// Mitsubishi GX Developer project: PLC_PCO520L2   PLC: Q06UDEH   RS485 Communication Modbus RTU

PROGRAM SP790_RS
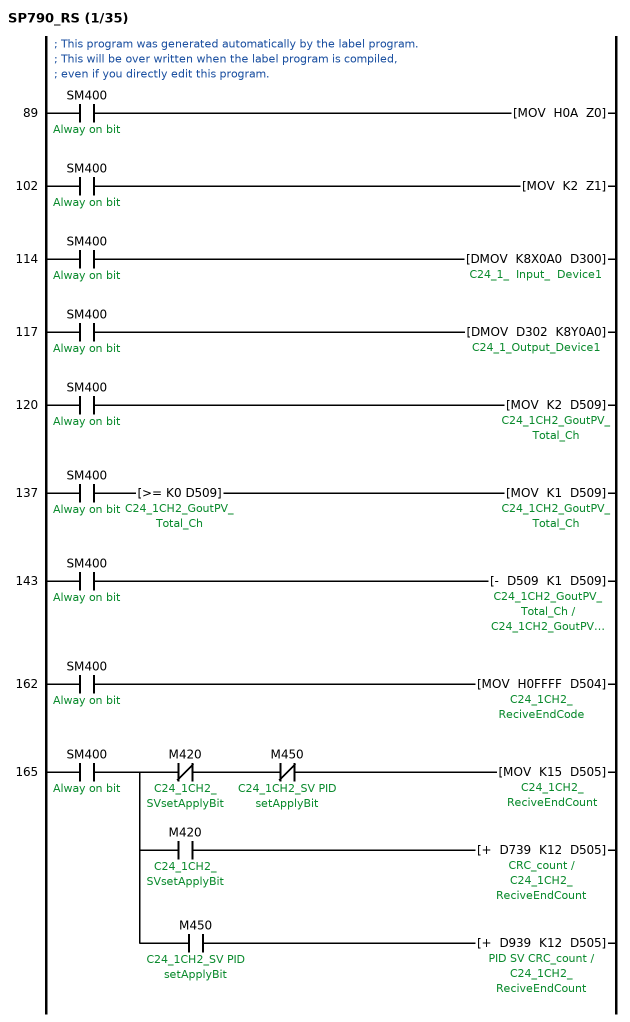
; This program was generated automatically by the label program.
; This will be over written when the label program is compiled,
; even if you directly edit this program.
89    LD      SM400  ; Alway on bit
      MOV     H0A Z0
        [note] Module IO Number
102   LD      SM400  ; Alway on bit
      MOV     K2 Z1
        [note] Channel Number
114   LD      SM400  ; Alway on bit
      DMOV    K8X0A0 D300  ; CH1 Transmission normal completi / C24_1_  Input_  Device1
117   LD      SM400  ; Alway on bit
      DMOV    D302 K8Y0A0  ; C24_1_Output_Device1 / CH1 Transmission request
120   LD      SM400  ; Alway on bit
      MOV     K2 D509  ; C24_1CH2_GoutPV_Total_Ch
        [note] Controller Channel Count
137   LD      SM400  ; Alway on bit
      AND>=   K0 D509  ; C24_1CH2_GoutPV_Total_Ch
      MOV     K1 D509
143   LD      SM400  ; Alway on bit
      -       D509 K1 D509
        [note] Controller Channel Count
162   LD      SM400  ; Alway on bit
      MOV     H0FFFF D504  ; C24_1CH2_ReciveEndCode
165   LD      SM400  ; Alway on bit
      MPS
      ANI     M420  ; C24_1CH2_SVsetApplyBit
      ANI     M450  ; C24_1CH2_SV PID setApplyBit
      MOV     K15 D505  ; C24_1CH2_ReciveEndCount
      MRD
      AND     M420  ; C24_1CH2_SVsetApplyBit
      +       D739 K12 D505  ; CRC_count
      MPP
      AND     M450  ; C24_1CH2_SV PID setApplyBit
      +       D939 K12 D505  ; PID SV CRC_count
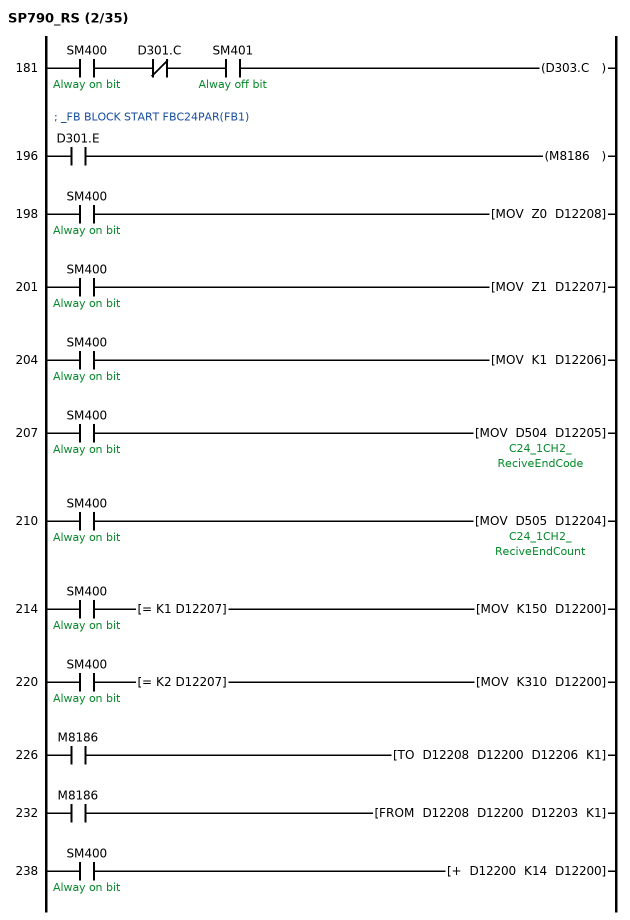
181   LD      SM400  ; Alway on bit
      ANI     D301.C
      AND     SM401  ; Alway off bit
      OUT     D303.C
        [note] System汲沥檬扁拳
; _FB BLOCK START FBC24PAR(FB1)
196   LD      D301.E
      OUT     M8186
198   LD      SM400  ; Alway on bit
      MOV     Z0 D12208
201   LD      SM400  ; Alway on bit
      MOV     Z1 D12207
204   LD      SM400  ; Alway on bit
      MOV     K1 D12206
207   LD      SM400  ; Alway on bit
      MOV     D504 D12205
210   LD      SM400  ; Alway on bit
      MOV     D505 D12204
; FB START
214   LD      SM400  ; Alway on bit
      AND=    K1 D12207
      MOV     K150 D12200
220   LD      SM400  ; Alway on bit
      AND=    K2 D12207
      MOV     K310 D12200
226   LD      M8186
      TO      D12208 D12200 D12206 K1
232   LD      M8186
      FROM    D12208 D12200 D12203 K1
238   LD      SM400  ; Alway on bit
      +       D12200 K14 D12200
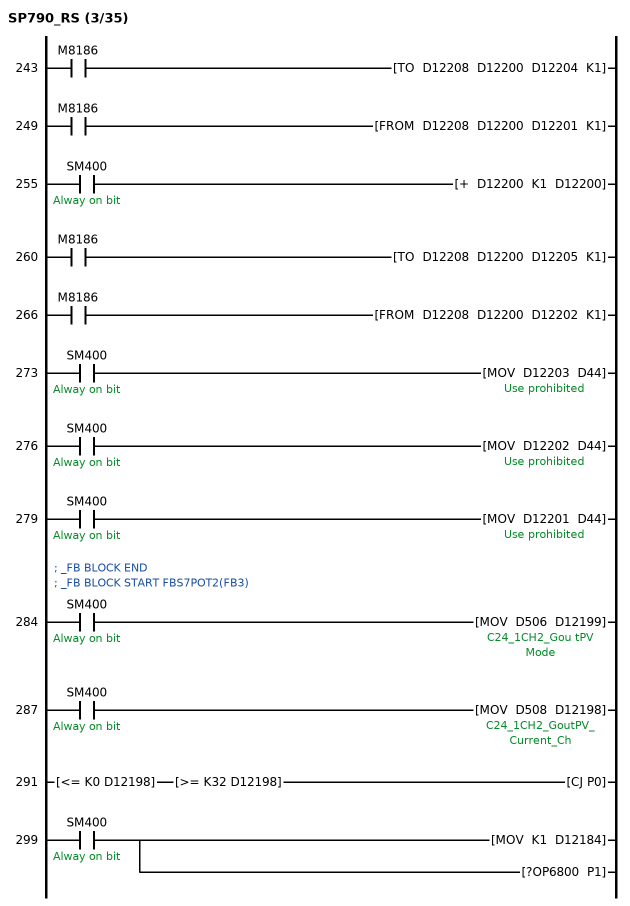
243   LD      M8186
      TO      D12208 D12200 D12204 K1
249   LD      M8186
      FROM    D12208 D12200 D12201 K1
255   LD      SM400  ; Alway on bit
      +       D12200 K1 D12200
260   LD      M8186
      TO      D12208 D12200 D12205 K1
266   LD      M8186
      FROM    D12208 D12200 D12202 K1
; FB END
273   LD      SM400  ; Alway on bit
      MOV     D12203 D44  ; Use prohibited
276   LD      SM400  ; Alway on bit
      MOV     D12202 D44
279   LD      SM400  ; Alway on bit
      MOV     D12201 D44
; _FB BLOCK END
; _FB BLOCK START FBS7POT2(FB3)
284   LD      SM400  ; Alway on bit
      MOV     D506 D12199  ; C24_1CH2_Gou tPV Mode
287   LD      SM400  ; Alway on bit
      MOV     D508 D12198  ; C24_1CH2_GoutPV_Current_Ch
; FB START
291   LD<=    K0 D12198
      AND>=   K32 D12198
      CJ      P0
299   LD      SM400  ; Alway on bit
      MOV     K1 D12184
      ?OP6800 P1
      P0
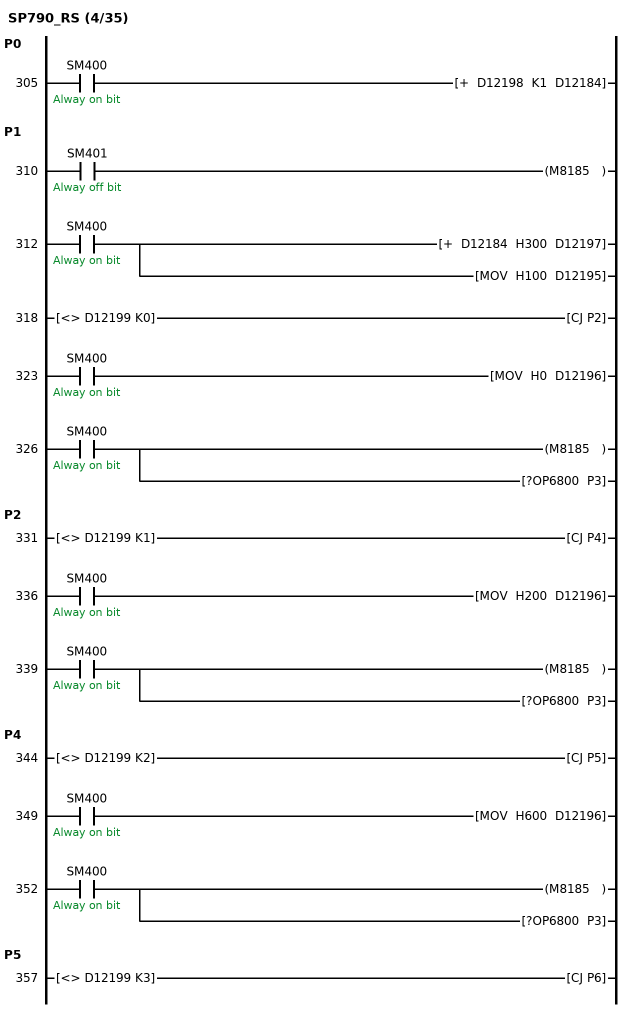
305   LD      SM400  ; Alway on bit
      +       D12198 K1 D12184
      P1
310   LD      SM401  ; Alway off bit
      OUT     M8185
312   LD      SM400  ; Alway on bit
      +       D12184 H300 D12197
      MOV     H100 D12195
318   LD<>    D12199 K0
      CJ      P2
323   LD      SM400  ; Alway on bit
      MOV     H0 D12196
326   LD      SM400  ; Alway on bit
      OUT     M8185
      ?OP6800 P3
      P2
331   LD<>    D12199 K1
      CJ      P4
336   LD      SM400  ; Alway on bit
      MOV     H200 D12196
339   LD      SM400  ; Alway on bit
      OUT     M8185
      ?OP6800 P3
      P4
344   LD<>    D12199 K2
      CJ      P5
349   LD      SM400  ; Alway on bit
      MOV     H600 D12196
352   LD      SM400  ; Alway on bit
      OUT     M8185
      ?OP6800 P3
      P5
357   LD<>    D12199 K3
      CJ      P6
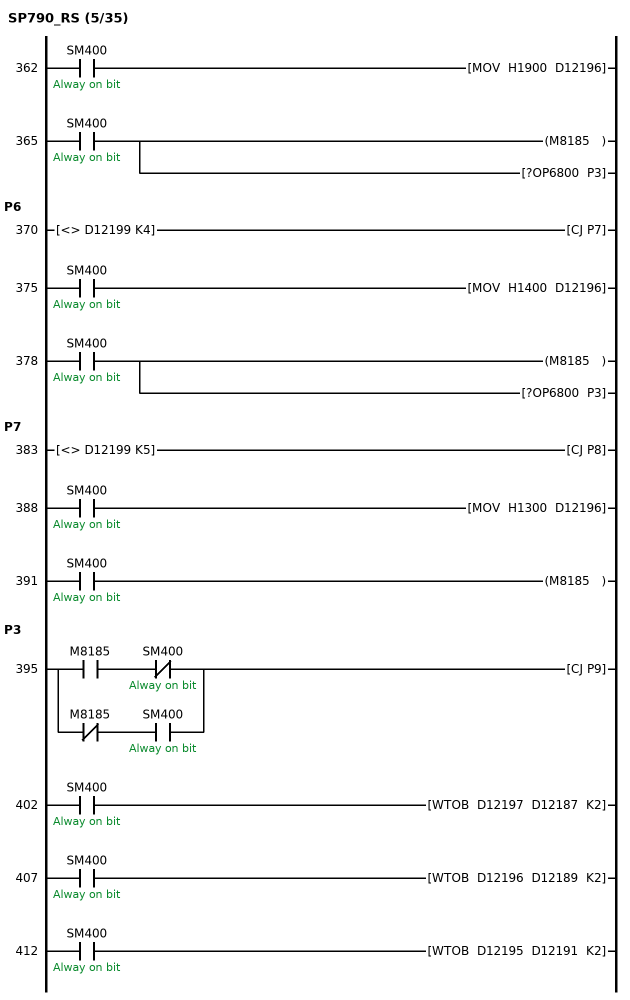
362   LD      SM400  ; Alway on bit
      MOV     H1900 D12196
365   LD      SM400  ; Alway on bit
      OUT     M8185
      ?OP6800 P3
      P6
370   LD<>    D12199 K4
      CJ      P7
375   LD      SM400  ; Alway on bit
      MOV     H1400 D12196
378   LD      SM400  ; Alway on bit
      OUT     M8185
      ?OP6800 P3
      P7
383   LD<>    D12199 K5
      CJ      P8
388   LD      SM400  ; Alway on bit
      MOV     H1300 D12196
391   LD      SM400  ; Alway on bit
      OUT     M8185
      P8
      P3
395   LD      M8185
      ANI     SM400  ; Alway on bit
      LDI     M8185
      AND     SM400  ; Alway on bit
      ORB
      CJ      P9
402   LD      SM400  ; Alway on bit
      WTOB    D12197 D12187 K2
407   LD      SM400  ; Alway on bit
      WTOB    D12196 D12189 K2
412   LD      SM400  ; Alway on bit
      WTOB    D12195 D12191 K2
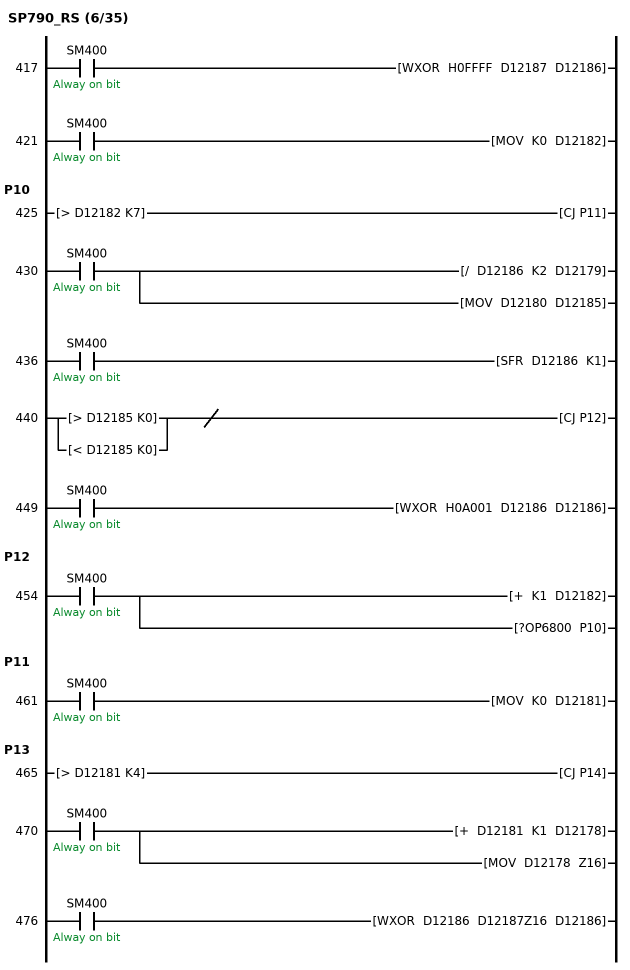
417   LD      SM400  ; Alway on bit
      WXOR    H0FFFF D12187 D12186
421   LD      SM400  ; Alway on bit
      MOV     K0 D12182
      P10
425   LD>     D12182 K7
      CJ      P11
430   LD      SM400  ; Alway on bit
      /       D12186 K2 D12179
      MOV     D12180 D12185
436   LD      SM400  ; Alway on bit
      SFR     D12186 K1
440   LD>     D12185 K0
      OR<     D12185 K0
      INV
      CJ      P12
449   LD      SM400  ; Alway on bit
      WXOR    H0A001 D12186 D12186
      P12
454   LD      SM400  ; Alway on bit
      +       K1 D12182
      ?OP6800 P10
      P11
461   LD      SM400  ; Alway on bit
      MOV     K0 D12181
      P13
465   LD>     D12181 K4
      CJ      P14
470   LD      SM400  ; Alway on bit
      +       D12181 K1 D12178
      MOV     D12178 Z16
476   LD      SM400  ; Alway on bit
      WXOR    D12186 D12187Z16 D12186
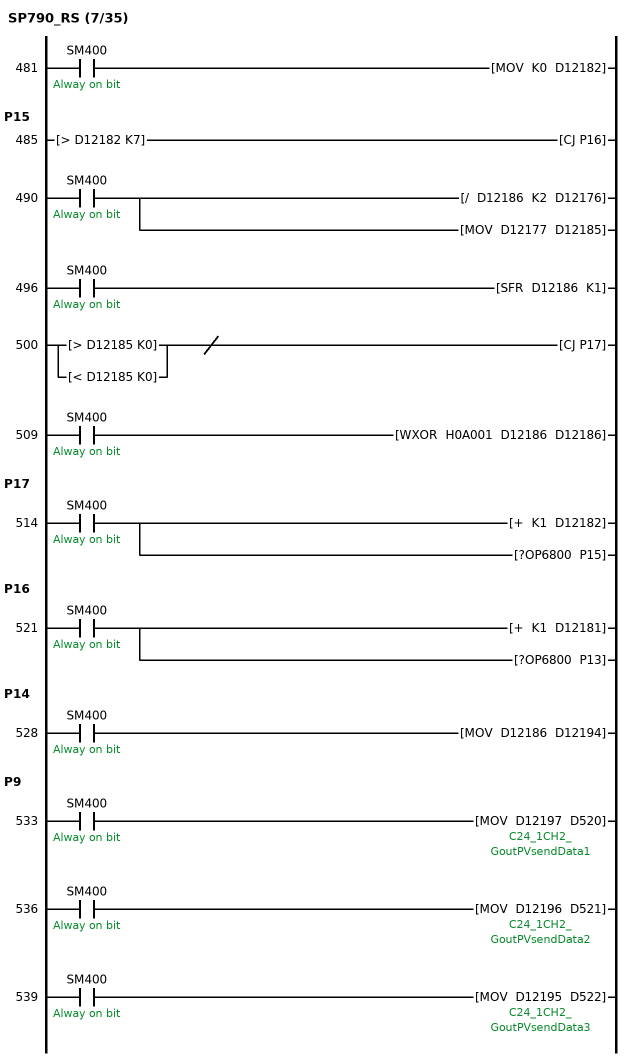
481   LD      SM400  ; Alway on bit
      MOV     K0 D12182
      P15
485   LD>     D12182 K7
      CJ      P16
490   LD      SM400  ; Alway on bit
      /       D12186 K2 D12176
      MOV     D12177 D12185
496   LD      SM400  ; Alway on bit
      SFR     D12186 K1
500   LD>     D12185 K0
      OR<     D12185 K0
      INV
      CJ      P17
509   LD      SM400  ; Alway on bit
      WXOR    H0A001 D12186 D12186
      P17
514   LD      SM400  ; Alway on bit
      +       K1 D12182
      ?OP6800 P15
      P16
521   LD      SM400  ; Alway on bit
      +       K1 D12181
      ?OP6800 P13
      P14
528   LD      SM400  ; Alway on bit
      MOV     D12186 D12194
      P9
; FB END
533   LD      SM400  ; Alway on bit
      MOV     D12197 D520  ; C24_1CH2_GoutPVsendData1
536   LD      SM400  ; Alway on bit
      MOV     D12196 D521  ; C24_1CH2_GoutPVsendData2
539   LD      SM400  ; Alway on bit
      MOV     D12195 D522  ; C24_1CH2_GoutPVsendData3
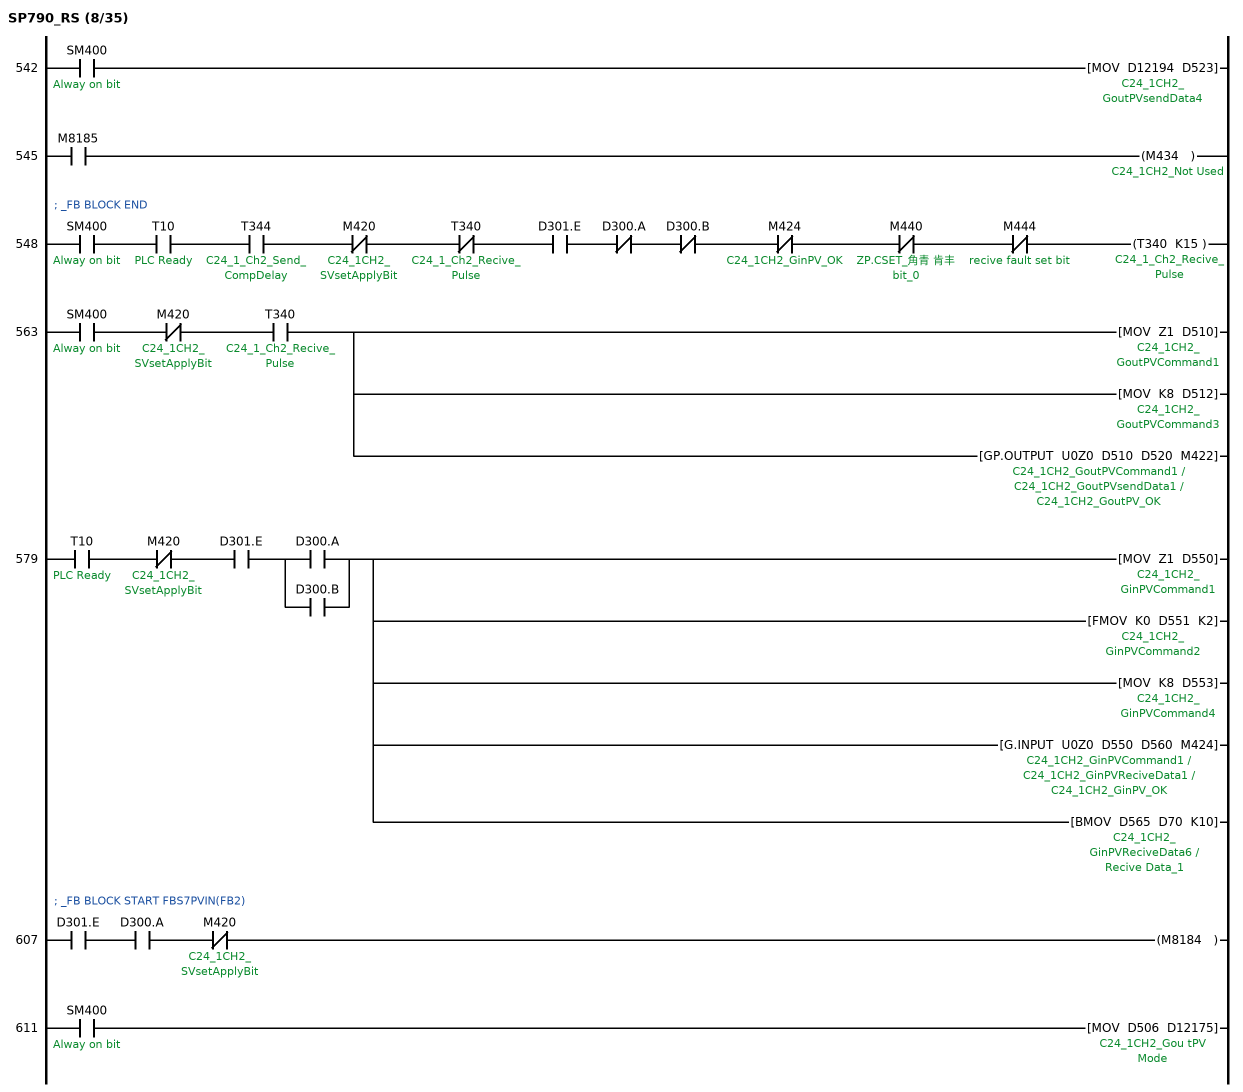
542   LD      SM400  ; Alway on bit
      MOV     D12194 D523  ; C24_1CH2_GoutPVsendData4
545   LD      M8185
      OUT     M434  ; C24_1CH2_Not Used
; _FB BLOCK END
548   LD      SM400  ; Alway on bit
      AND     T10  ; PLC Ready
      AND     T344  ; C24_1_Ch2_Send_CompDelay
      ANI     M420  ; C24_1CH2_SVsetApplyBit
      ANI     T340  ; C24_1_Ch2_Recive_Pulse
      AND     D301.E
      ANI     D300.A
      ANI     D300.B
      ANI     M424  ; C24_1CH2_GinPV_OK
      ANI     M440  ; ZP.CSET_角青 肯丰 bit_0
      ANI     M444  ; recive fault set bit
      OUTH    T340 K15  ; C24_1_Ch2_Recive_Pulse
563   LD      SM400  ; Alway on bit
      ANI     M420  ; C24_1CH2_SVsetApplyBit
      AND     T340  ; C24_1_Ch2_Recive_Pulse
      MOV     Z1 D510  ; C24_1CH2_GoutPVCommand1
      MOV     K8 D512  ; C24_1CH2_GoutPVCommand3
      GP.OUTPUT U0Z0 D510 D520 M422  ; C24_1CH2_GoutPV_OK
579   LD      T10  ; PLC Ready
      ANI     M420  ; C24_1CH2_SVsetApplyBit
      AND     D301.E
      LD      D300.A
      OR      D300.B
      ANB
      MOV     Z1 D550  ; C24_1CH2_GinPVCommand1
      FMOV    K0 D551 K2  ; C24_1CH2_GinPVCommand2
      MOV     K8 D553  ; C24_1CH2_GinPVCommand4
      G.INPUT U0Z0 D550 D560 M424  ; C24_1CH2_GinPVReciveData1
      BMOV    D565 D70 K10  ; C24_1CH2_GinPVReciveData6 / Recive Data_1
; _FB BLOCK START FBS7PVIN(FB2)
607   LD      D301.E
      AND     D300.A
      ANI     M420  ; C24_1CH2_SVsetApplyBit
      OUT     M8184
611   LD      SM400  ; Alway on bit
      MOV     D506 D12175
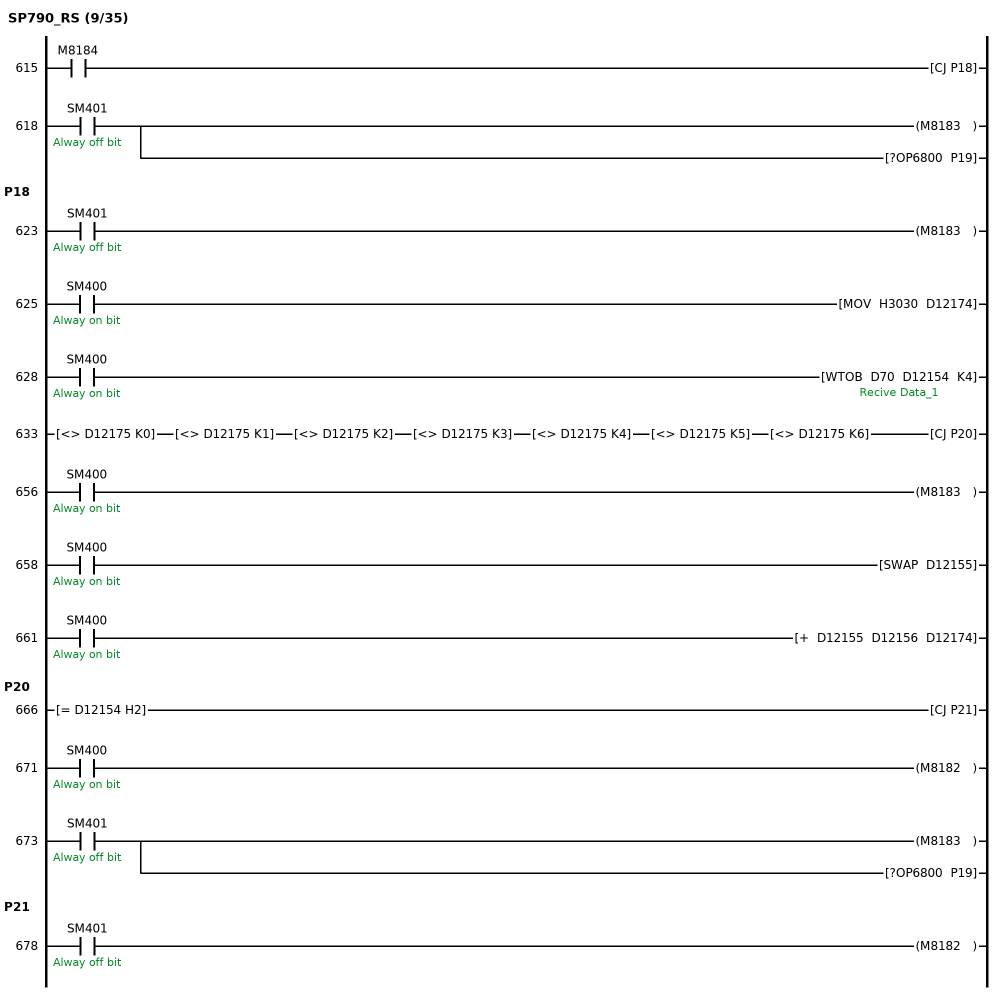
; FB START
615   LD      M8184
      CJ      P18
618   LD      SM401  ; Alway off bit
      OUT     M8183
      ?OP6800 P19
      P18
623   LD      SM401  ; Alway off bit
      OUT     M8183
625   LD      SM400  ; Alway on bit
      MOV     H3030 D12174
628   LD      SM400  ; Alway on bit
      WTOB    D70 D12154 K4
633   LD<>    D12175 K0
      AND<>   D12175 K1
      AND<>   D12175 K2
      AND<>   D12175 K3
      AND<>   D12175 K4
      AND<>   D12175 K5
      AND<>   D12175 K6
      CJ      P20
656   LD      SM400  ; Alway on bit
      OUT     M8183
658   LD      SM400  ; Alway on bit
      SWAP    D12155
661   LD      SM400  ; Alway on bit
      +       D12155 D12156 D12174
      P20
666   LD=     D12154 H2
      CJ      P21
671   LD      SM400  ; Alway on bit
      OUT     M8182
673   LD      SM401  ; Alway off bit
      OUT     M8183
      ?OP6800 P19
      P21
678   LD      SM401  ; Alway off bit
      OUT     M8182
      P19
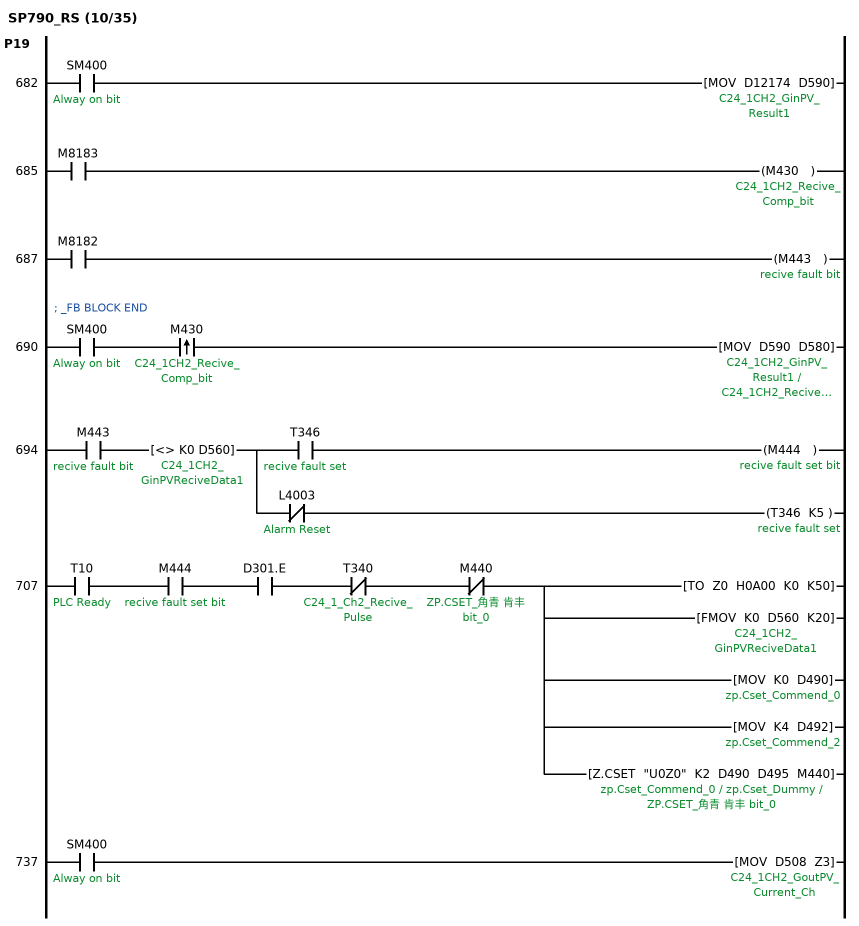
; FB END
682   LD      SM400  ; Alway on bit
      MOV     D12174 D590  ; C24_1CH2_GinPV_Result1
685   LD      M8183
      OUT     M430  ; C24_1CH2_Recive_Comp_bit
687   LD      M8182
      OUT     M443  ; recive fault bit
; _FB BLOCK END
690   LD      SM400  ; Alway on bit
      ANDP    M430  ; C24_1CH2_Recive_Comp_bit
      MOV     D590 D580  ; C24_1CH2_Recive_Value_1
694   LD      M443  ; recive fault bit
      AND<>   K0 D560  ; C24_1CH2_GinPVReciveData1
      MPS
      AND     T346  ; recive fault set
      OUT     M444  ; recive fault set bit
      MPP
      ANI     L4003  ; Alarm Reset
      OUT     T346 K5  ; recive fault set
707   LD      T10  ; PLC Ready
      AND     M444  ; recive fault set bit
      AND     D301.E
      ANI     T340  ; C24_1_Ch2_Recive_Pulse
      ANI     M440  ; ZP.CSET_角青 肯丰 bit_0
      TO      Z0 H0A00 K0 K50
      FMOV    K0 D560 K20
      MOV     K0 D490  ; zp.Cset_Commend_0
      MOV     K4 D492  ; zp.Cset_Commend_2
      Z.CSET  "U0Z0" K2 D490 D495 M440  ; zp.Cset_Dummy
737   LD      SM400  ; Alway on bit
      MOV     D508 Z3
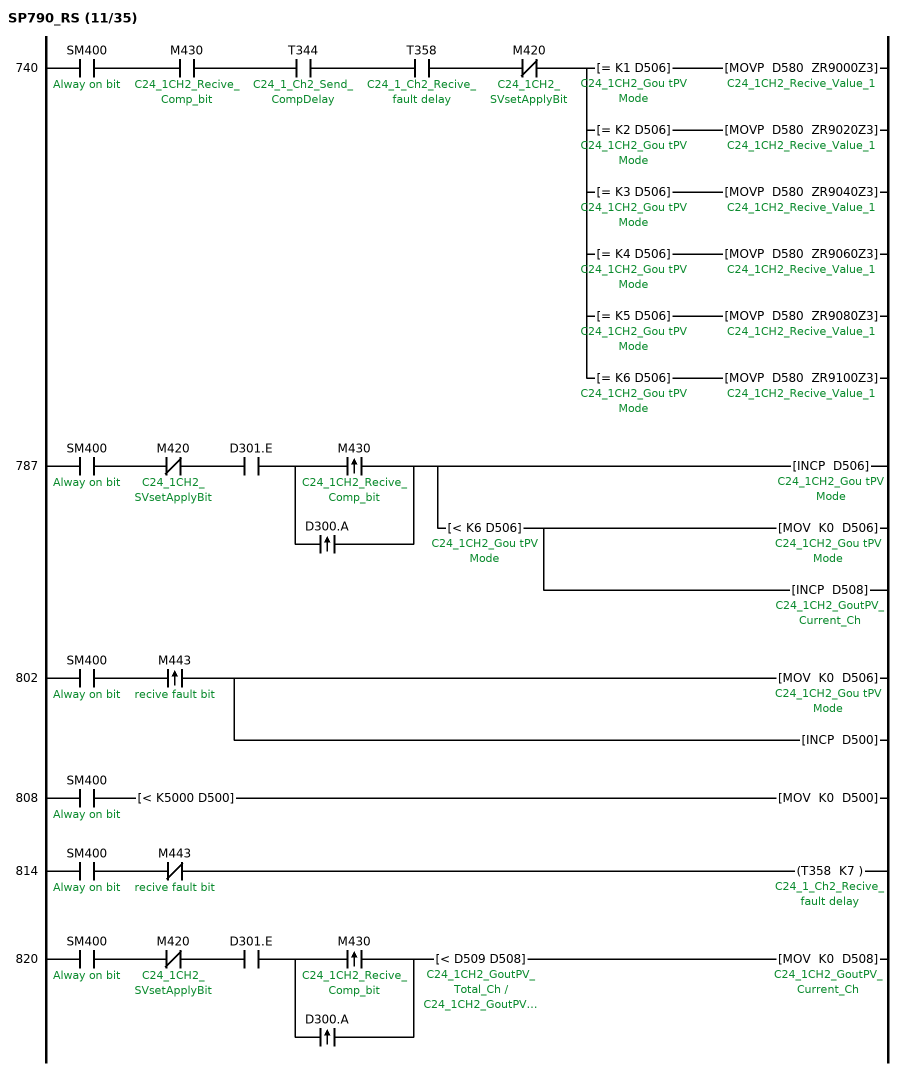
740   LD      SM400  ; Alway on bit
      AND     M430  ; C24_1CH2_Recive_Comp_bit
      AND     T344  ; C24_1_Ch2_Send_CompDelay
      AND     T358  ; C24_1_Ch2_Recive_fault delay
      ANI     M420  ; C24_1CH2_SVsetApplyBit
      MPS
      AND=    K1 D506  ; C24_1CH2_Gou tPV Mode
      MOVP    D580 ZR9000Z3
      MRD
      AND=    K2 D506  ; C24_1CH2_Gou tPV Mode
      MOVP    D580 ZR9020Z3
      MRD
      AND=    K3 D506  ; C24_1CH2_Gou tPV Mode
      MOVP    D580 ZR9040Z3
      MRD
      AND=    K4 D506  ; C24_1CH2_Gou tPV Mode
      MOVP    D580 ZR9060Z3
      MRD
      AND=    K5 D506  ; C24_1CH2_Gou tPV Mode
      MOVP    D580 ZR9080Z3
      MPP
      AND=    K6 D506  ; C24_1CH2_Gou tPV Mode
      MOVP    D580 ZR9100Z3
787   LD      SM400  ; Alway on bit
      ANI     M420  ; C24_1CH2_SVsetApplyBit
      AND     D301.E
      LDP     M430  ; C24_1CH2_Recive_Comp_bit
      ORP     D300.A
      ANB
      INCP    D506
      AND<    K6 D506  ; C24_1CH2_Gou tPV Mode
      MOV     K0 D506
      INCP    D508
802   LD      SM400  ; Alway on bit
      ANDP    M443  ; recive fault bit
      MOV     K0 D506
      INCP    D500
808   LD      SM400  ; Alway on bit
      AND<    K5000 D500
      MOV     K0 D500
814   LD      SM400  ; Alway on bit
      ANI     M443  ; recive fault bit
      OUT     T358 K7  ; C24_1_Ch2_Recive_fault delay
820   LD      SM400  ; Alway on bit
      ANI     M420  ; C24_1CH2_SVsetApplyBit
      AND     D301.E
      LDP     M430  ; C24_1CH2_Recive_Comp_bit
      ORP     D300.A
      ANB
      AND<    D509 D508  ; C24_1CH2_GoutPV_Total_Ch / C24_1CH2_GoutPV_Current_Ch
      MOV     K0 D508
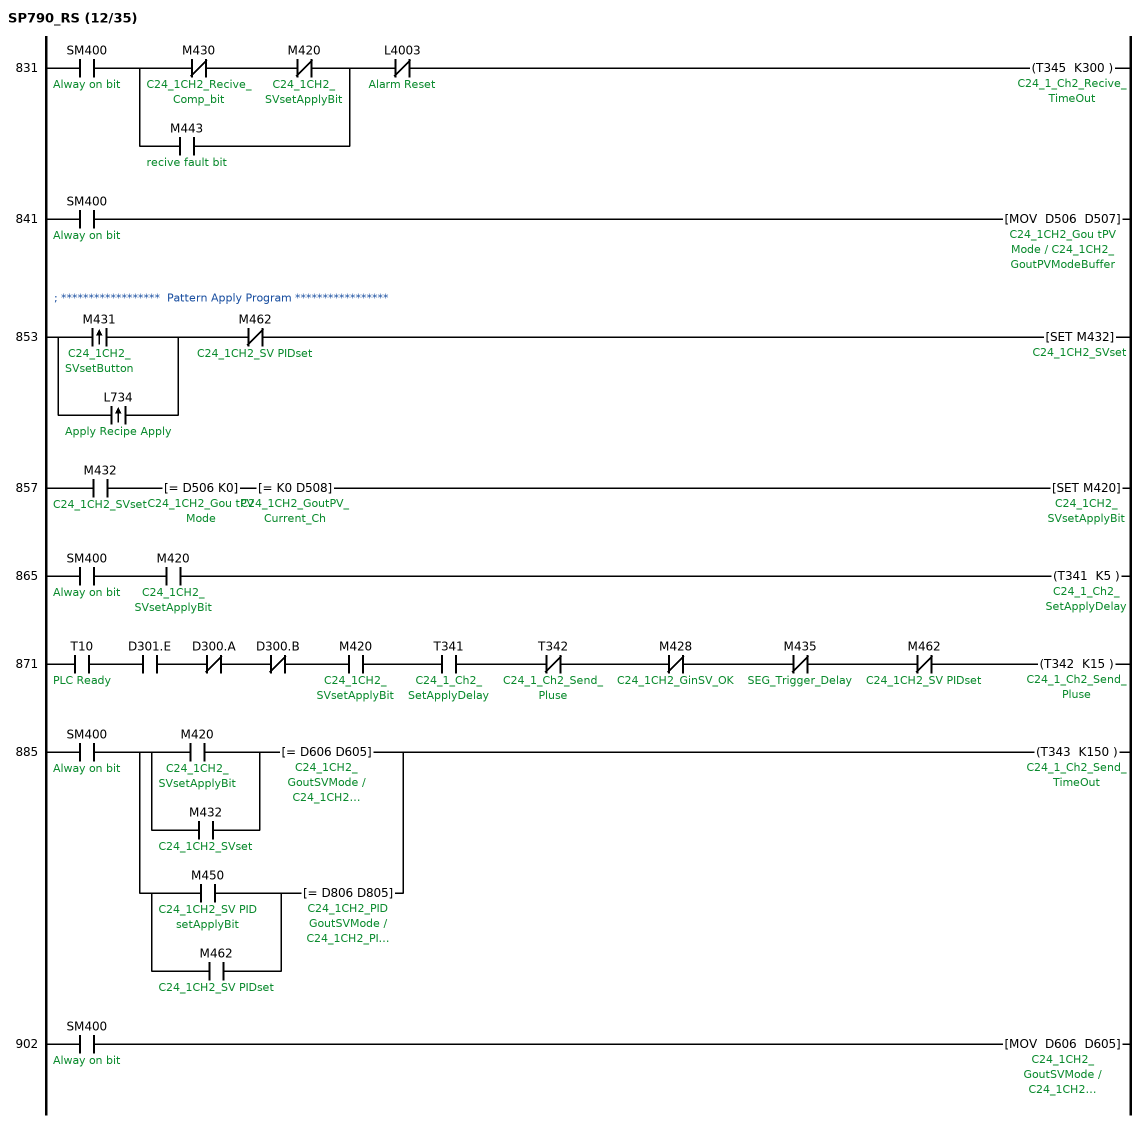
831   LD      SM400  ; Alway on bit
      LDI     M430  ; C24_1CH2_Recive_Comp_bit
      ANI     M420  ; C24_1CH2_SVsetApplyBit
      OR      M443  ; recive fault bit
      ANB
      ANI     L4003  ; Alarm Reset
      OUT     T345 K300  ; C24_1_Ch2_Recive_TimeOut
841   LD      SM400  ; Alway on bit
      MOV     D506 D507  ; C24_1CH2_GoutPVModeBuffer
; 
; 
; 
; 
; ******************  Pattern Apply Program *****************
853   LDP     M431  ; C24_1CH2_SVsetButton
      ORP     L734  ; Apply Recipe Apply
      ANI     M462  ; C24_1CH2_SV PIDset
      SET     M432  ; C24_1CH2_SVset
857   LD      M432  ; C24_1CH2_SVset
      AND=    D506 K0  ; C24_1CH2_Gou tPV Mode
      AND=    K0 D508  ; C24_1CH2_GoutPV_Current_Ch
      SET     M420  ; C24_1CH2_SVsetApplyBit
865   LD      SM400  ; Alway on bit
      AND     M420  ; C24_1CH2_SVsetApplyBit
      OUT     T341 K5  ; C24_1_Ch2_SetApplyDelay
871   LD      T10  ; PLC Ready
      AND     D301.E
      ANI     D300.A
      ANI     D300.B
      AND     M420  ; C24_1CH2_SVsetApplyBit
      AND     T341  ; C24_1_Ch2_SetApplyDelay
      ANI     T342  ; C24_1_Ch2_Send_Pluse
      ANI     M428  ; C24_1CH2_GinSV_OK
      ANI     M435  ; SEG_Trigger_Delay
      ANI     M462  ; C24_1CH2_SV PIDset
      OUTH    T342 K15  ; C24_1_Ch2_Send_Pluse
885   LD      SM400  ; Alway on bit
      LD      M420  ; C24_1CH2_SVsetApplyBit
      OR      M432  ; C24_1CH2_SVset
      AND=    D606 D605  ; C24_1CH2_GoutSVMode / C24_1CH2_ModeBuffer
      LD      M450  ; C24_1CH2_SV PID setApplyBit
      OR      M462  ; C24_1CH2_SV PIDset
      AND=    D806 D805  ; C24_1CH2_PID GoutSVMode / C24_1CH2_PID ModeBuffer
      ORB
      ANB
      OUT     T343 K150  ; C24_1_Ch2_Send_TimeOut
902   LD      SM400  ; Alway on bit
      MOV     D606 D605
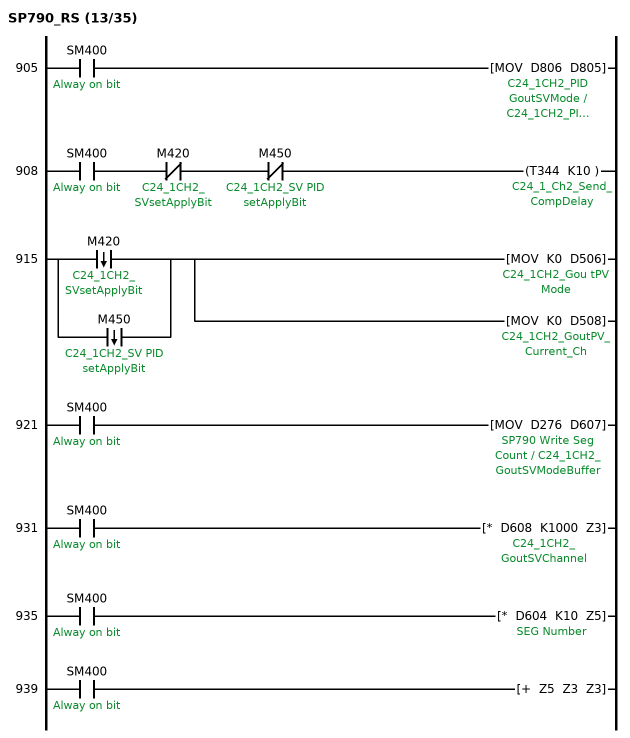
905   LD      SM400  ; Alway on bit
      MOV     D806 D805
908   LD      SM400  ; Alway on bit
      ANI     M420  ; C24_1CH2_SVsetApplyBit
      ANI     M450  ; C24_1CH2_SV PID setApplyBit
      OUT     T344 K10  ; C24_1_Ch2_Send_CompDelay
915   LDF     M420  ; C24_1CH2_SVsetApplyBit
      ORF     M450  ; C24_1CH2_SV PID setApplyBit
      MOV     K0 D506
      MOV     K0 D508
921   LD      SM400  ; Alway on bit
      MOV     D276 D607  ; SP790 Write Seg Count / C24_1CH2_GoutSVModeBuffer
        [note] Seg Count
931   LD      SM400  ; Alway on bit
      *       D608 K1000 Z3  ; C24_1CH2_GoutSVChannel
935   LD      SM400  ; Alway on bit
      *       D604 K10 Z5  ; SEG Number
939   LD      SM400  ; Alway on bit
      +       Z5 Z3 Z3
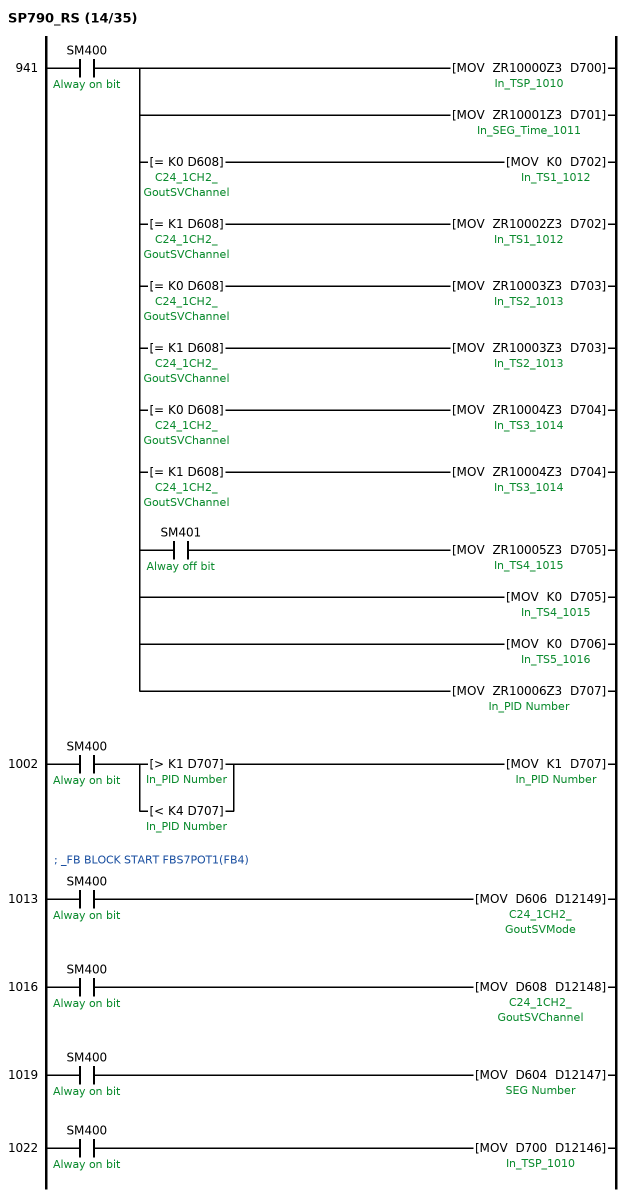
941   LD      SM400  ; Alway on bit
      MOV     ZR10000Z3 D700  ; In_TSP_1010
      MOV     ZR10001Z3 D701  ; In_SEG_Time_1011
      MPS
      AND=    K0 D608  ; C24_1CH2_GoutSVChannel
      MOV     K0 D702  ; In_TS1_1012
      MRD
      AND=    K1 D608  ; C24_1CH2_GoutSVChannel
      MOV     ZR10002Z3 D702
      MRD
      AND=    K0 D608  ; C24_1CH2_GoutSVChannel
      MOV     ZR10003Z3 D703  ; In_TS2_1013
      MRD
      AND=    K1 D608  ; C24_1CH2_GoutSVChannel
      MOV     ZR10003Z3 D703
      MRD
      AND=    K0 D608  ; C24_1CH2_GoutSVChannel
      MOV     ZR10004Z3 D704  ; In_TS3_1014
      MRD
      AND=    K1 D608  ; C24_1CH2_GoutSVChannel
      MOV     ZR10004Z3 D704
      MRD
      AND     SM401  ; Alway off bit
      MOV     ZR10005Z3 D705  ; In_TS4_1015
      MPP
      MOV     K0 D705
      MOV     K0 D706  ; In_TS5_1016
      MOV     ZR10006Z3 D707  ; In_PID Number
1002  LD      SM400  ; Alway on bit
      LD>     K1 D707  ; In_PID Number
      OR<     K4 D707  ; In_PID Number
      ANB
      MOV     K1 D707
; _FB BLOCK START FBS7POT1(FB4)
1013  LD      SM400  ; Alway on bit
      MOV     D606 D12149
1016  LD      SM400  ; Alway on bit
      MOV     D608 D12148
1019  LD      SM400  ; Alway on bit
      MOV     D604 D12147
1022  LD      SM400  ; Alway on bit
      MOV     D700 D12146
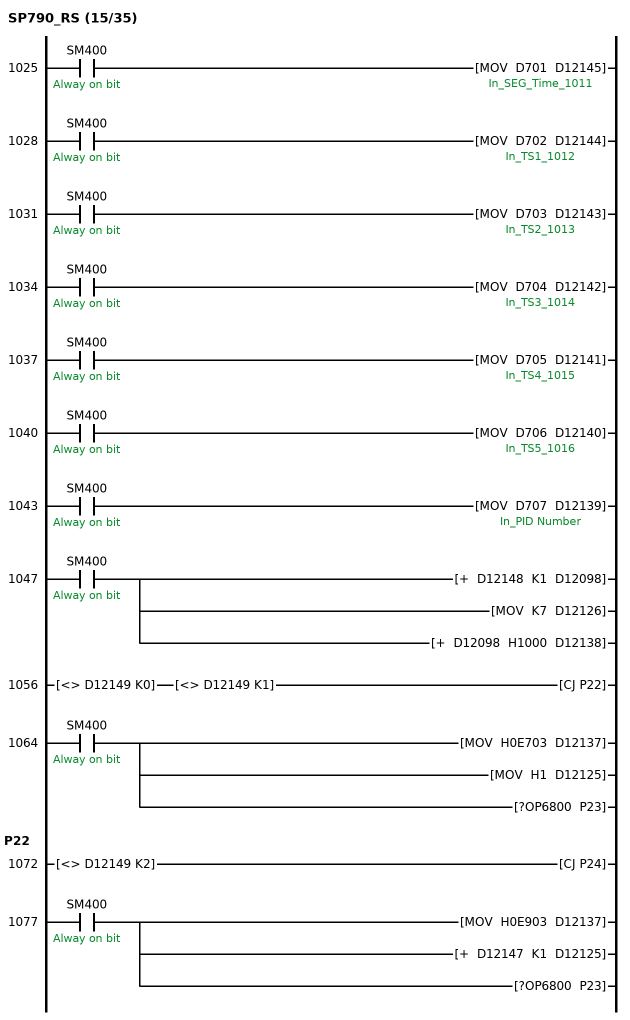
1025  LD      SM400  ; Alway on bit
      MOV     D701 D12145
1028  LD      SM400  ; Alway on bit
      MOV     D702 D12144
1031  LD      SM400  ; Alway on bit
      MOV     D703 D12143
1034  LD      SM400  ; Alway on bit
      MOV     D704 D12142
1037  LD      SM400  ; Alway on bit
      MOV     D705 D12141
1040  LD      SM400  ; Alway on bit
      MOV     D706 D12140
1043  LD      SM400  ; Alway on bit
      MOV     D707 D12139
; FB START
1047  LD      SM400  ; Alway on bit
      +       D12148 K1 D12098
      MOV     K7 D12126
      +       D12098 H1000 D12138
1056  LD<>    D12149 K0
      AND<>   D12149 K1
      CJ      P22
1064  LD      SM400  ; Alway on bit
      MOV     H0E703 D12137
      MOV     H1 D12125
      ?OP6800 P23
      P22
1072  LD<>    D12149 K2
      CJ      P24
1077  LD      SM400  ; Alway on bit
      MOV     H0E903 D12137
      +       D12147 K1 D12125
      ?OP6800 P23
      P24
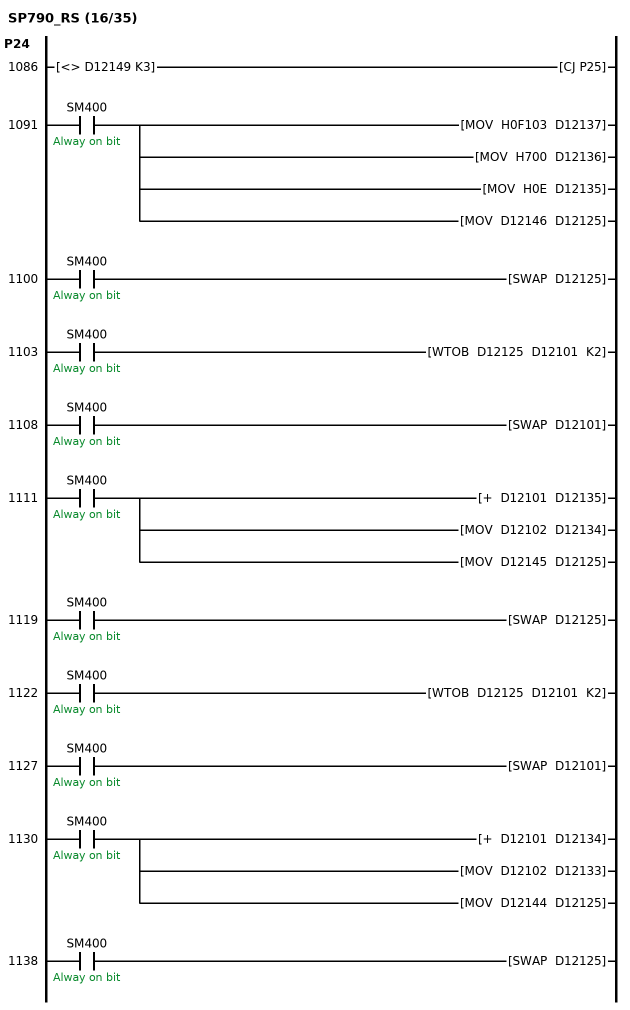
1086  LD<>    D12149 K3
      CJ      P25
1091  LD      SM400  ; Alway on bit
      MOV     H0F103 D12137
      MOV     H700 D12136
      MOV     H0E D12135
      MOV     D12146 D12125
1100  LD      SM400  ; Alway on bit
      SWAP    D12125
1103  LD      SM400  ; Alway on bit
      WTOB    D12125 D12101 K2
1108  LD      SM400  ; Alway on bit
      SWAP    D12101
1111  LD      SM400  ; Alway on bit
      +       D12101 D12135
      MOV     D12102 D12134
      MOV     D12145 D12125
1119  LD      SM400  ; Alway on bit
      SWAP    D12125
1122  LD      SM400  ; Alway on bit
      WTOB    D12125 D12101 K2
1127  LD      SM400  ; Alway on bit
      SWAP    D12101
1130  LD      SM400  ; Alway on bit
      +       D12101 D12134
      MOV     D12102 D12133
      MOV     D12144 D12125
1138  LD      SM400  ; Alway on bit
      SWAP    D12125
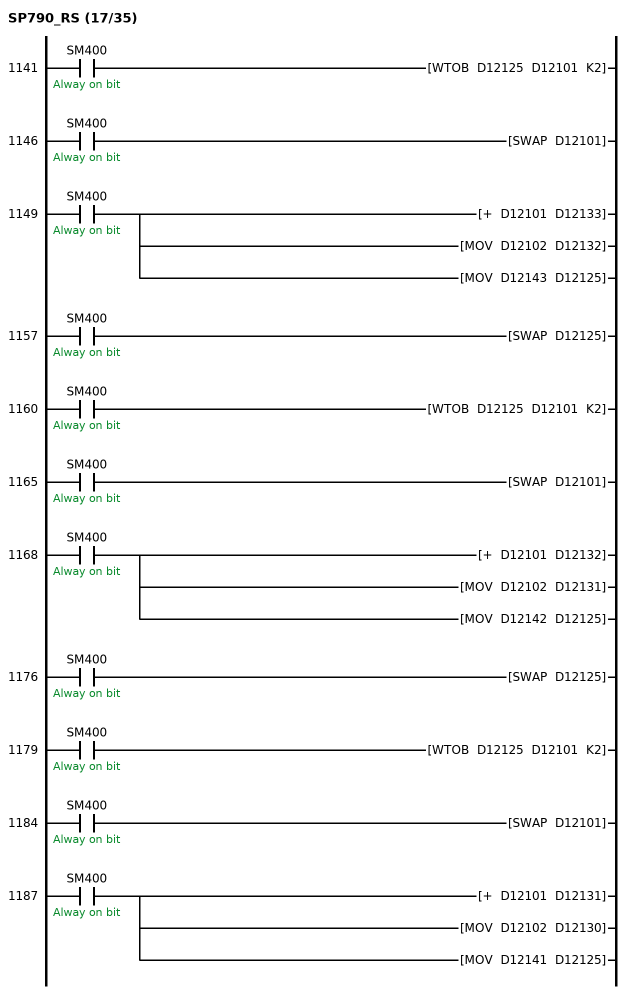
1141  LD      SM400  ; Alway on bit
      WTOB    D12125 D12101 K2
1146  LD      SM400  ; Alway on bit
      SWAP    D12101
1149  LD      SM400  ; Alway on bit
      +       D12101 D12133
      MOV     D12102 D12132
      MOV     D12143 D12125
1157  LD      SM400  ; Alway on bit
      SWAP    D12125
1160  LD      SM400  ; Alway on bit
      WTOB    D12125 D12101 K2
1165  LD      SM400  ; Alway on bit
      SWAP    D12101
1168  LD      SM400  ; Alway on bit
      +       D12101 D12132
      MOV     D12102 D12131
      MOV     D12142 D12125
1176  LD      SM400  ; Alway on bit
      SWAP    D12125
1179  LD      SM400  ; Alway on bit
      WTOB    D12125 D12101 K2
1184  LD      SM400  ; Alway on bit
      SWAP    D12101
1187  LD      SM400  ; Alway on bit
      +       D12101 D12131
      MOV     D12102 D12130
      MOV     D12141 D12125
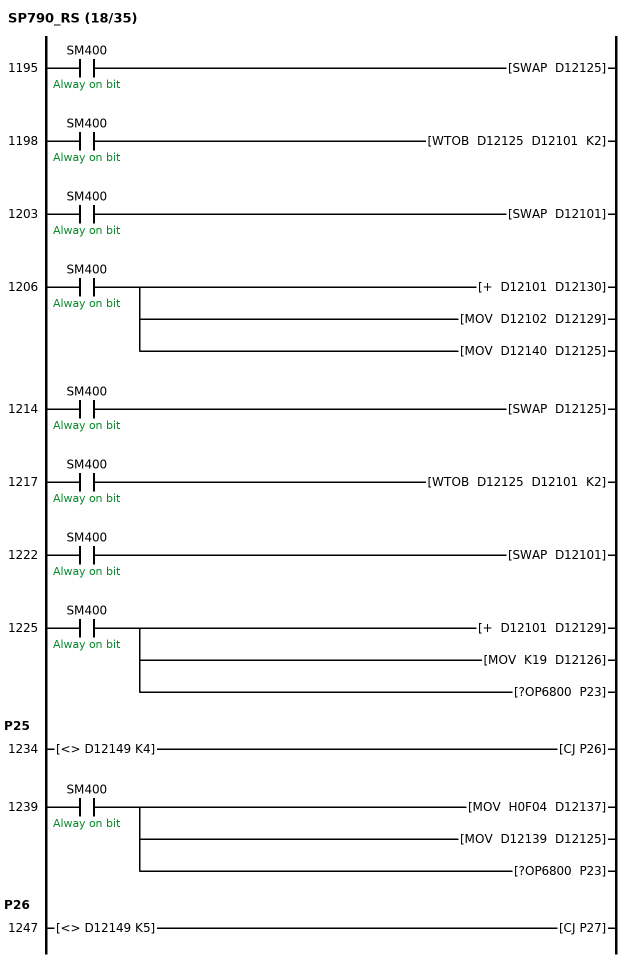
1195  LD      SM400  ; Alway on bit
      SWAP    D12125
1198  LD      SM400  ; Alway on bit
      WTOB    D12125 D12101 K2
1203  LD      SM400  ; Alway on bit
      SWAP    D12101
1206  LD      SM400  ; Alway on bit
      +       D12101 D12130
      MOV     D12102 D12129
      MOV     D12140 D12125
1214  LD      SM400  ; Alway on bit
      SWAP    D12125
1217  LD      SM400  ; Alway on bit
      WTOB    D12125 D12101 K2
1222  LD      SM400  ; Alway on bit
      SWAP    D12101
1225  LD      SM400  ; Alway on bit
      +       D12101 D12129
      MOV     K19 D12126
      ?OP6800 P23
      P25
1234  LD<>    D12149 K4
      CJ      P26
1239  LD      SM400  ; Alway on bit
      MOV     H0F04 D12137
      MOV     D12139 D12125
      ?OP6800 P23
      P26
1247  LD<>    D12149 K5
      CJ      P27
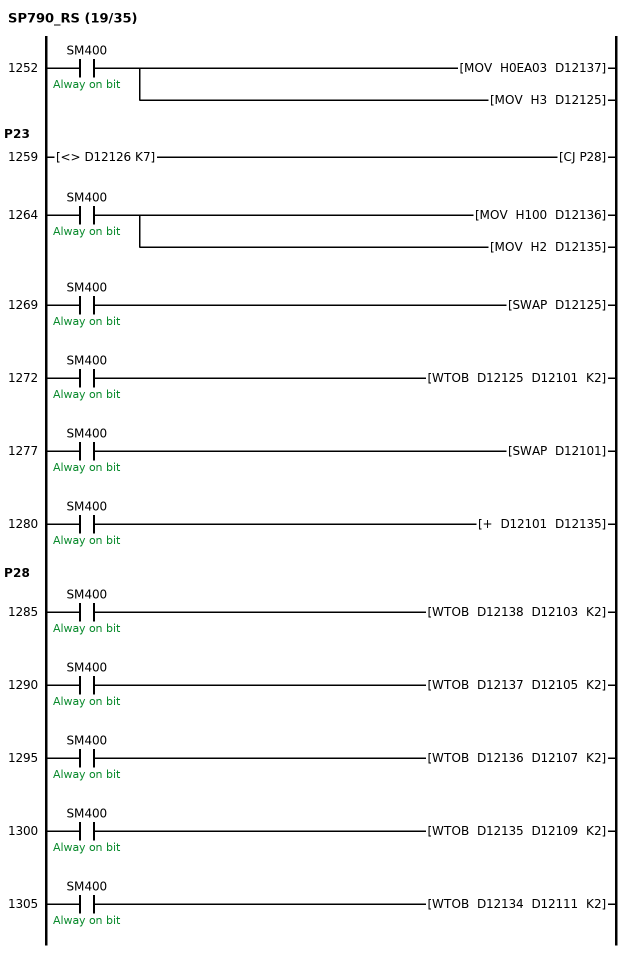
1252  LD      SM400  ; Alway on bit
      MOV     H0EA03 D12137
      MOV     H3 D12125
      P27
      P23
1259  LD<>    D12126 K7
      CJ      P28
1264  LD      SM400  ; Alway on bit
      MOV     H100 D12136
      MOV     H2 D12135
1269  LD      SM400  ; Alway on bit
      SWAP    D12125
1272  LD      SM400  ; Alway on bit
      WTOB    D12125 D12101 K2
1277  LD      SM400  ; Alway on bit
      SWAP    D12101
1280  LD      SM400  ; Alway on bit
      +       D12101 D12135
      P28
1285  LD      SM400  ; Alway on bit
      WTOB    D12138 D12103 K2
1290  LD      SM400  ; Alway on bit
      WTOB    D12137 D12105 K2
1295  LD      SM400  ; Alway on bit
      WTOB    D12136 D12107 K2
1300  LD      SM400  ; Alway on bit
      WTOB    D12135 D12109 K2
1305  LD      SM400  ; Alway on bit
      WTOB    D12134 D12111 K2
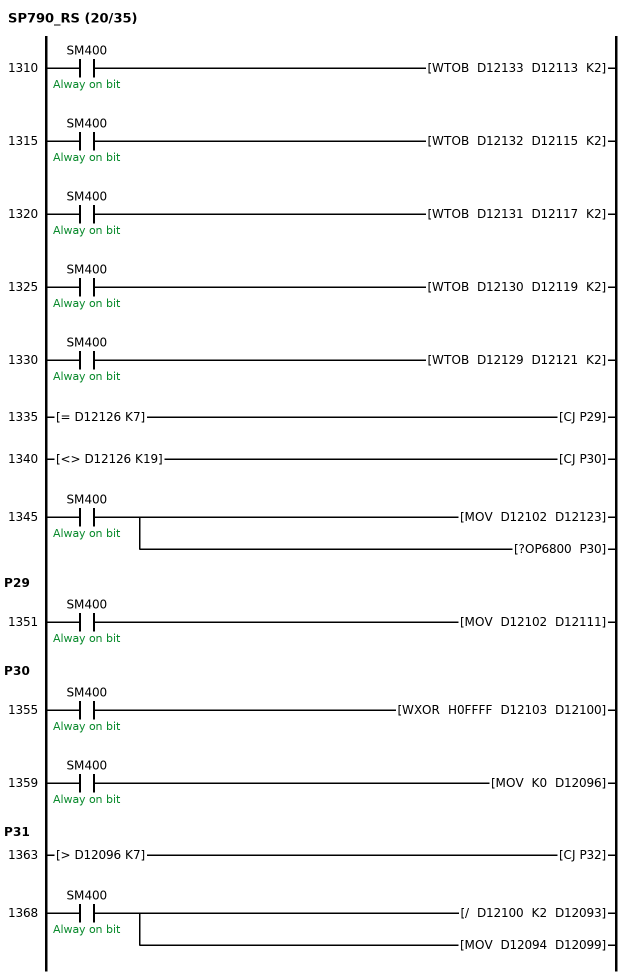
1310  LD      SM400  ; Alway on bit
      WTOB    D12133 D12113 K2
1315  LD      SM400  ; Alway on bit
      WTOB    D12132 D12115 K2
1320  LD      SM400  ; Alway on bit
      WTOB    D12131 D12117 K2
1325  LD      SM400  ; Alway on bit
      WTOB    D12130 D12119 K2
1330  LD      SM400  ; Alway on bit
      WTOB    D12129 D12121 K2
1335  LD=     D12126 K7
      CJ      P29
1340  LD<>    D12126 K19
      CJ      P30
1345  LD      SM400  ; Alway on bit
      MOV     D12102 D12123
      ?OP6800 P30
      P29
1351  LD      SM400  ; Alway on bit
      MOV     D12102 D12111
      P30
1355  LD      SM400  ; Alway on bit
      WXOR    H0FFFF D12103 D12100
1359  LD      SM400  ; Alway on bit
      MOV     K0 D12096
      P31
1363  LD>     D12096 K7
      CJ      P32
1368  LD      SM400  ; Alway on bit
      /       D12100 K2 D12093
      MOV     D12094 D12099
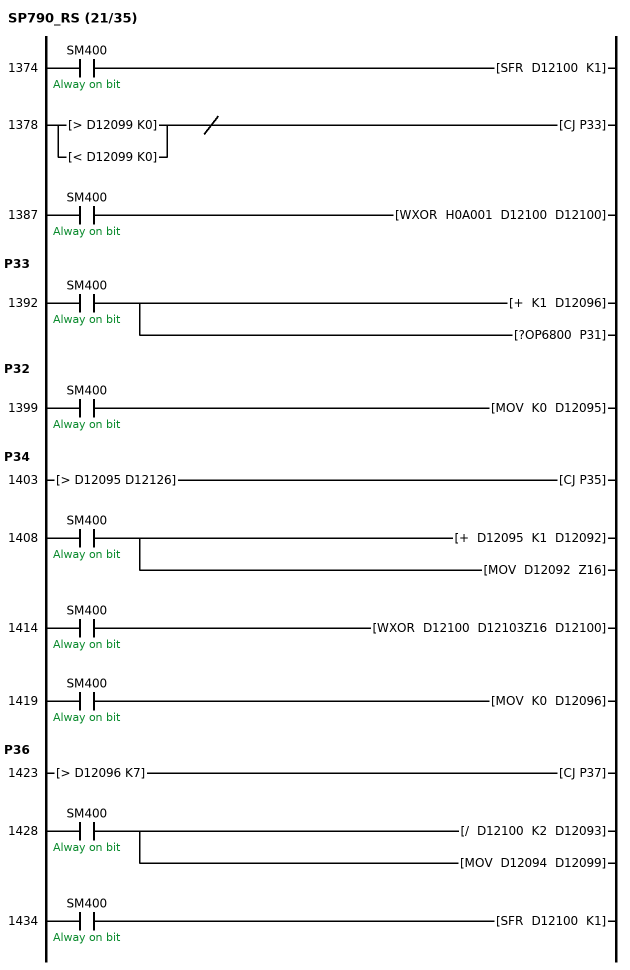
1374  LD      SM400  ; Alway on bit
      SFR     D12100 K1
1378  LD>     D12099 K0
      OR<     D12099 K0
      INV
      CJ      P33
1387  LD      SM400  ; Alway on bit
      WXOR    H0A001 D12100 D12100
      P33
1392  LD      SM400  ; Alway on bit
      +       K1 D12096
      ?OP6800 P31
      P32
1399  LD      SM400  ; Alway on bit
      MOV     K0 D12095
      P34
1403  LD>     D12095 D12126
      CJ      P35
1408  LD      SM400  ; Alway on bit
      +       D12095 K1 D12092
      MOV     D12092 Z16
1414  LD      SM400  ; Alway on bit
      WXOR    D12100 D12103Z16 D12100
1419  LD      SM400  ; Alway on bit
      MOV     K0 D12096
      P36
1423  LD>     D12096 K7
      CJ      P37
1428  LD      SM400  ; Alway on bit
      /       D12100 K2 D12093
      MOV     D12094 D12099
1434  LD      SM400  ; Alway on bit
      SFR     D12100 K1
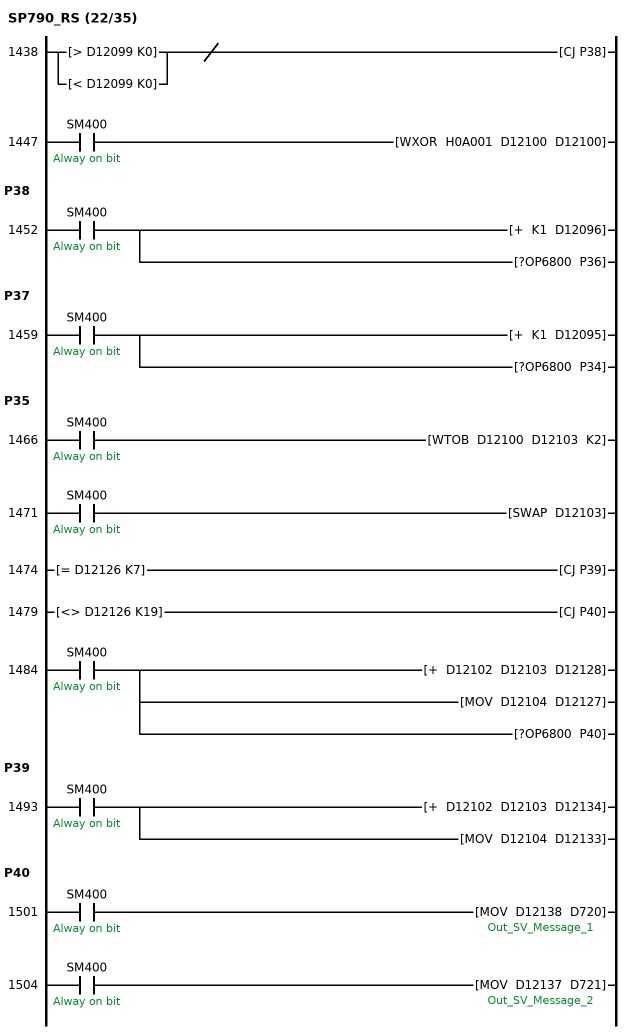
1438  LD>     D12099 K0
      OR<     D12099 K0
      INV
      CJ      P38
1447  LD      SM400  ; Alway on bit
      WXOR    H0A001 D12100 D12100
      P38
1452  LD      SM400  ; Alway on bit
      +       K1 D12096
      ?OP6800 P36
      P37
1459  LD      SM400  ; Alway on bit
      +       K1 D12095
      ?OP6800 P34
      P35
1466  LD      SM400  ; Alway on bit
      WTOB    D12100 D12103 K2
1471  LD      SM400  ; Alway on bit
      SWAP    D12103
1474  LD=     D12126 K7
      CJ      P39
1479  LD<>    D12126 K19
      CJ      P40
1484  LD      SM400  ; Alway on bit
      +       D12102 D12103 D12128
      MOV     D12104 D12127
      ?OP6800 P40
      P39
1493  LD      SM400  ; Alway on bit
      +       D12102 D12103 D12134
      MOV     D12104 D12133
      P40
; FB END
1501  LD      SM400  ; Alway on bit
      MOV     D12138 D720  ; Out_SV_Message_1
1504  LD      SM400  ; Alway on bit
      MOV     D12137 D721  ; Out_SV_Message_2
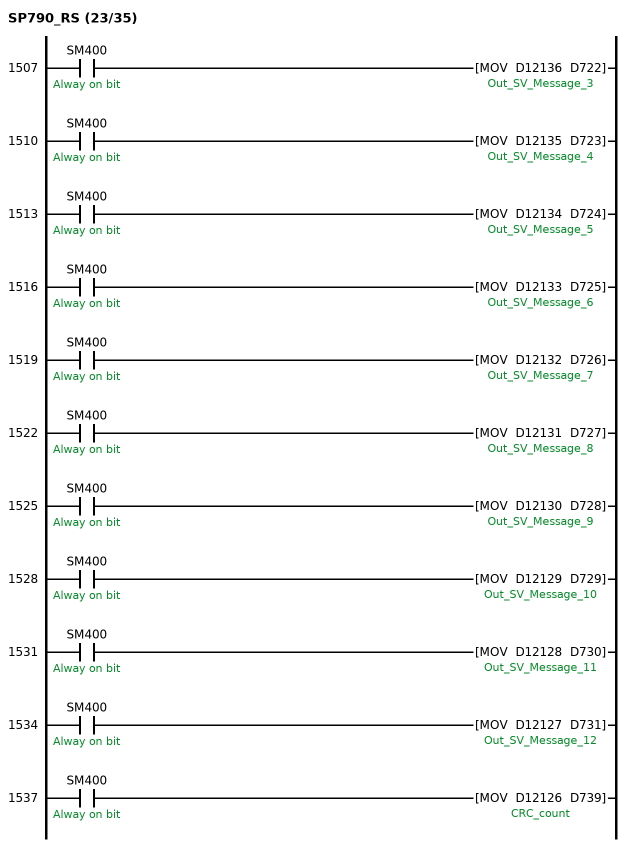
1507  LD      SM400  ; Alway on bit
      MOV     D12136 D722  ; Out_SV_Message_3
1510  LD      SM400  ; Alway on bit
      MOV     D12135 D723  ; Out_SV_Message_4
1513  LD      SM400  ; Alway on bit
      MOV     D12134 D724  ; Out_SV_Message_5
1516  LD      SM400  ; Alway on bit
      MOV     D12133 D725  ; Out_SV_Message_6
1519  LD      SM400  ; Alway on bit
      MOV     D12132 D726  ; Out_SV_Message_7
1522  LD      SM400  ; Alway on bit
      MOV     D12131 D727  ; Out_SV_Message_8
1525  LD      SM400  ; Alway on bit
      MOV     D12130 D728  ; Out_SV_Message_9
1528  LD      SM400  ; Alway on bit
      MOV     D12129 D729  ; Out_SV_Message_10
1531  LD      SM400  ; Alway on bit
      MOV     D12128 D730  ; Out_SV_Message_11
1534  LD      SM400  ; Alway on bit
      MOV     D12127 D731  ; Out_SV_Message_12
1537  LD      SM400  ; Alway on bit
      MOV     D12126 D739
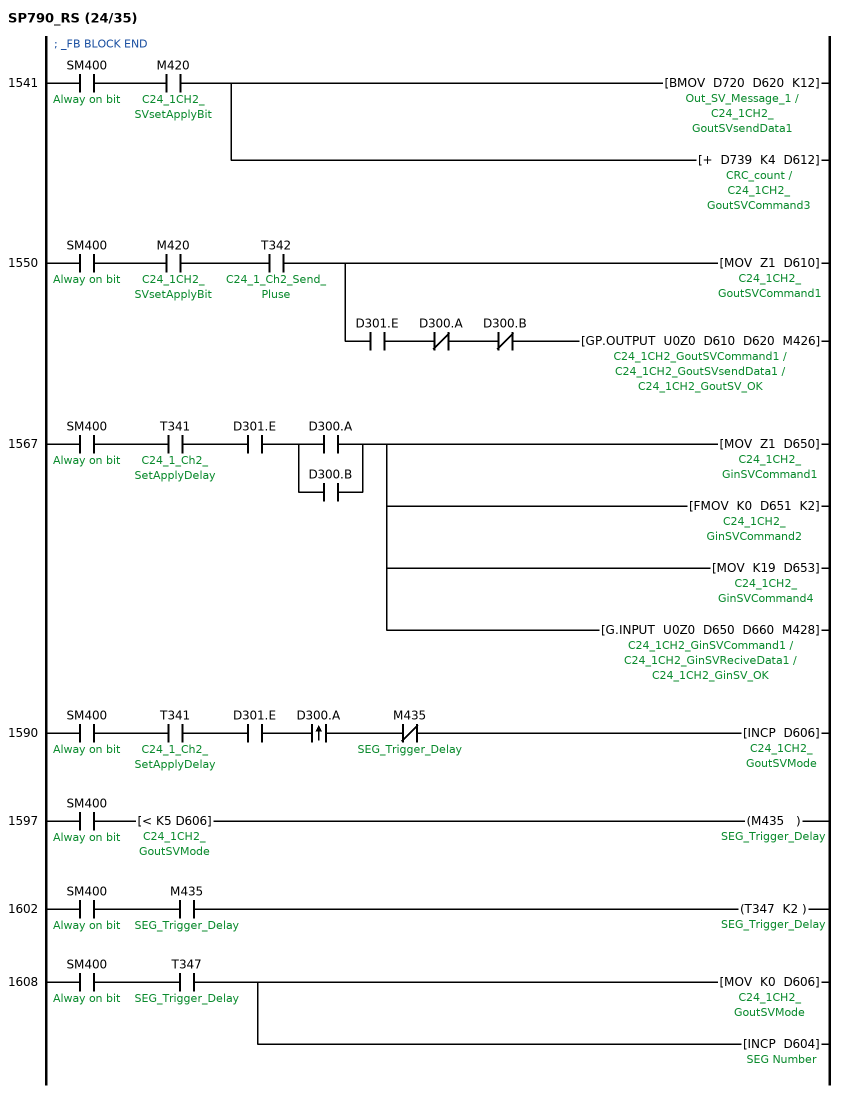
; _FB BLOCK END
1541  LD      SM400  ; Alway on bit
      AND     M420  ; C24_1CH2_SVsetApplyBit
      BMOV    D720 D620 K12  ; C24_1CH2_GoutSVsendData1
      +       D739 K4 D612  ; C24_1CH2_GoutSVCommand3
1550  LD      SM400  ; Alway on bit
      AND     M420  ; C24_1CH2_SVsetApplyBit
      AND     T342  ; C24_1_Ch2_Send_Pluse
      MOV     Z1 D610  ; C24_1CH2_GoutSVCommand1
      AND     D301.E
      ANI     D300.A
      ANI     D300.B
      GP.OUTPUT U0Z0 D610 D620 M426  ; C24_1CH2_GoutSV_OK
1567  LD      SM400  ; Alway on bit
      AND     T341  ; C24_1_Ch2_SetApplyDelay
      AND     D301.E
      LD      D300.A
      OR      D300.B
      ANB
      MOV     Z1 D650  ; C24_1CH2_GinSVCommand1
      FMOV    K0 D651 K2  ; C24_1CH2_GinSVCommand2
      MOV     K19 D653  ; C24_1CH2_GinSVCommand4
      G.INPUT U0Z0 D650 D660 M428  ; C24_1CH2_GinSVReciveData1
1590  LD      SM400  ; Alway on bit
      AND     T341  ; C24_1_Ch2_SetApplyDelay
      AND     D301.E
      ANDP    D300.A
      ANI     M435  ; SEG_Trigger_Delay
      INCP    D606
1597  LD      SM400  ; Alway on bit
      AND<    K5 D606  ; C24_1CH2_GoutSVMode
      OUT     M435  ; SEG_Trigger_Delay
1602  LD      SM400  ; Alway on bit
      AND     M435  ; SEG_Trigger_Delay
      OUT     T347 K2  ; SEG_Trigger_Delay
1608  LD      SM400  ; Alway on bit
      AND     T347  ; SEG_Trigger_Delay
      MOV     K0 D606
      INCP    D604
